FUNCTION_BLOCK HandshakeRequesterWSTRING (* Handshake pattern demo (WSTRING payload): Plug / Requester role *)
  (* Standard: 61499-2; Description: Copyright (c) 2026 Meisterschulen am Ostbahnhof This program and the accompanying materials are made available under the terms of the Eclipse Public License 2.0 which is available at https://www.eclipse.org/legal/epl-2.0/ SPDX-License-Identifier: EPL-2.0 *)
  (* Version 1.1, 2026-08-31, Franz Höpfinger, Meisterschulen am Ostbahnhof, HS.REQD/HS.CNFD/HS.INDD/HS.RSPD access syntax confirmed working in 4diac; ack payload moved to HandshakeConst::ACK_PAYLOAD (const/HandshakeConst.gcf) instead of a literal *)
  (* Version 1.0, 2026-08-31, Franz Höpfinger, Meisterschulen am Ostbahnhof, Handshake design pattern (IEC 61499 primer course, Module 6, Valeriy Vyatkin), demo Requester with WSTRING payload via EVENT_HS_WSTRING *)
  PACKAGE Meins::DesingPatterns::HandshakePattern;
  IMPORT Meins::DesingPatterns::HandshakePattern::const::HandshakeConst;
  (* Documentation:
  Requester ("client") side of the Handshake design pattern, data-carrying variant (IEC 61499 primer course, Module 6, Valeriy Vyatkin; adapter matches slide 48's generic "service" adapter).
   Uses adapter::events::Handshake::EVENT_HS_WSTRING as a Plug: on START it loads ReqPayload into HS.REQD and sends REQ; reports DONE (with CnfPayload) once the matching CNF comes back; whenever an unsolicited IND arrives it reads HS.INDD into IndPayload, answers with a fixed "ack" RSP and reports NOTIFIED.
   See HandshakePattern.md in this folder for the full write-up.
  *)
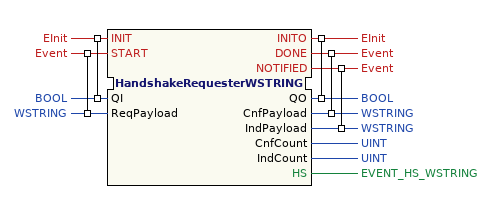
  EVENT_INPUT
    INIT : EInit WITH QI; (* Initialization Request *)
    START WITH ReqPayload; (* Demo: fire a REQ (with ReqPayload) towards the Responder *)
  END_EVENT
  EVENT_OUTPUT
    INITO : EInit WITH QO; (* Initialization Confirm *)
    DONE WITH CnfPayload; (* A CNF (with CnfPayload) was received for the last REQ *)
    NOTIFIED WITH IndPayload; (* An IND (with IndPayload) was received and answered with RSP *)
  END_EVENT
  VAR_INPUT
    QI : BOOL; (* Input event qualifier *)
    ReqPayload : WSTRING := "push,100"; (* Payload sent with the next REQ *)
  END_VAR
  VAR_OUTPUT
    QO : BOOL; (* Output event qualifier *)
    CnfPayload : WSTRING; (* Payload of the last received CNF *)
    IndPayload : WSTRING; (* Payload of the last received IND *)
    CnfCount : UINT; (* Number of CNF received (demo counter) *)
    IndCount : UINT; (* Number of IND received / RSP sent (demo counter) *)
  END_VAR
  PLUGS
    HS : adapter::events::Handshake::EVENT_HS_WSTRING; (* Handshake plug: sends REQ/RSP (+REQD/RSPD), receives CNF/IND (+CNFD/INDD) *)
  END_PLUGS
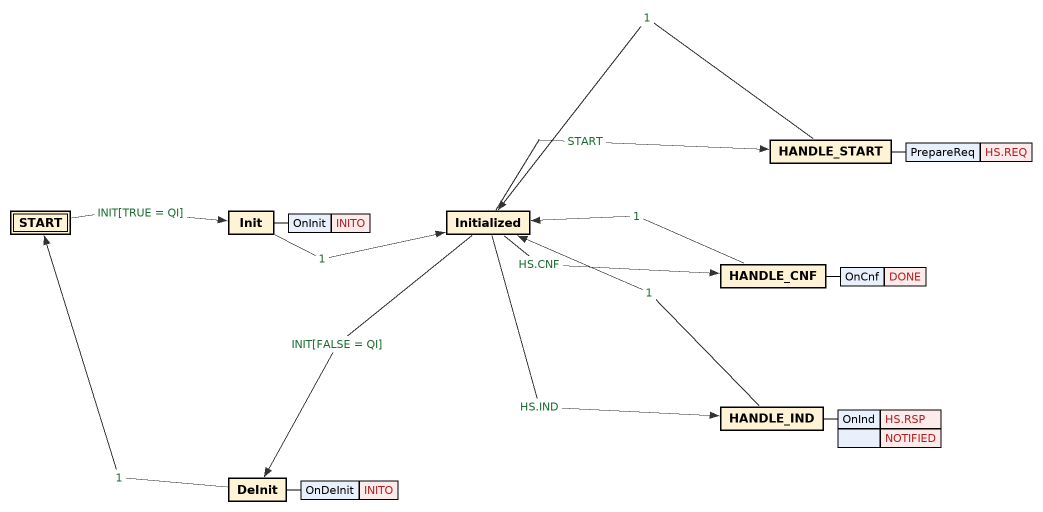
  EC_STATES
    START; (* Uninitialized *)
    Init : OnInit -> INITO; (* Initialization *)
    Initialized; (* Idle, ready to react *)
    DeInit : OnDeInit -> INITO; (* De-initialization *)
    HANDLE_START : PrepareReq -> HS.REQ; (* Prepare REQD and send a REQ *)
    HANDLE_CNF : OnCnf -> DONE; (* A CNF arrived, report DONE *)
    HANDLE_IND : OnInd -> HS.RSP, -> NOTIFIED; (* An IND arrived, answer with RSP and report NOTIFIED *)
  END_STATES
  EC_TRANSITIONS
    START TO Init := INIT[TRUE = QI];
    Init TO Initialized := 1;
    Initialized TO DeInit := INIT[FALSE = QI];
    DeInit TO START := 1;
    Initialized TO HANDLE_START := START;
    HANDLE_START TO Initialized := 1;
    Initialized TO HANDLE_CNF := HS.CNF;
    HANDLE_CNF TO Initialized := 1;
    Initialized TO HANDLE_IND := HS.IND;
    HANDLE_IND TO Initialized := 1;
  END_TRANSITIONS
  ALGORITHM OnInit IN ST: (* Reset demo counters/payloads *)
CnfCount := 0;
IndCount := 0;
CnfPayload := "";
IndPayload := "";
QO := QI;
  END_ALGORITHM
  ALGORITHM OnDeInit IN ST: (* De-initialize *)
QO := FALSE;
  END_ALGORITHM
  ALGORITHM PrepareReq IN ST: (* Load REQD from ReqPayload before HS.REQ fires *)
HS.REQD := ReqPayload;
  END_ALGORITHM
  ALGORITHM OnCnf IN ST: (* Read CNFD, count a received CNF *)
CnfPayload := HS.CNFD;
CnfCount := CnfCount + 1;
  END_ALGORITHM
  ALGORITHM OnInd IN ST: (* Read INDD, count a received IND, prepare RSPD *)
IndPayload := HS.INDD;
IndCount := IndCount + 1;
HS.RSPD := HandshakeConst::ACK_PAYLOAD;
  END_ALGORITHM
END_FUNCTION_BLOCK
